VAR_GLOBAL
	I_xTsEstopCH1					AT%I*: BOOL;
	I_xTsEstopCH2					AT%I*: BOOL;
	I_xTsE_Stop			 			AT%I*: BOOL;
	I_xTsCommErr					AT%I*: BOOL;
	I_xTsLightGridOK				AT%I*: BOOL;
	I_xTsFBErr						AT%I*: BOOL;
END_VAR

(* stored: Version 1.1.0.1, ProductVersion 3.1.4022.18
   GVL SAFETY_IN_GLV: Id {f89b2a94-5083-4808-bbe7-228b6775b654} *)
